(* PLC project Sem nome, Desconhecido Sem nome 1 *)
(* stored: creationDateTime 2025-09-02T10:17:35, modificationDateTime 2025-09-05T09:58:23 *)

PROGRAM program0
  VAR
    HighSensor AT %IX100.0 : BOOL;
    LowSensor AT %IX100.1 : BOOL;
    PalletSensor AT %IX100.2 : BOOL;
    Loaded AT %IX100.3 : BOOL;
    AtLeftEntry AT %IX100.4 : BOOL;
    AtLeftExit AT %IX100.5 : BOOL;
    AtRightEntry AT %IX100.6 : BOOL;
    AtRightExit AT %IX100.7 : BOOL;
    Start AT %IX100.8 : BOOL;
    Reset AT %IX100.9 : BOOL;
    Stop AT %IX100.10 : BOOL;
    EmergencyStop AT %IX100.11 : BOOL;
    Auto AT %IX100.12 : BOOL;
    ConveyorEntry AT %QX100.0 : BOOL;
    Load AT %QX100.1 : BOOL;
    Unload AT %QX100.2 : BOOL;
    TransferLeft AT %QX100.3 : BOOL;
    TransferRight AT %QX100.4 : BOOL;
    ConveyorLeft AT %QX100.5 : BOOL;
    ConveyorRight AT %QX100.6 : BOOL;
    StartLight AT %QX100.7 : BOOL;
    ResetLight AT %QX100.8 : BOOL;
    StopLight AT %QX100.9 : BOOL;
  END_VAR
  VAR
    MemoryRight : BOOL;
    MemoryLeft : BOOL;
  END_VAR
  VAR
    Counter AT %QW100 : INT;
  END_VAR
  VAR
    CTU0 : CTU;
  END_VAR
  VAR  (* added by the conversion: wires and edge detectors of the diagram *)
    R_TRIG1 : R_TRIG;
  END_VAR

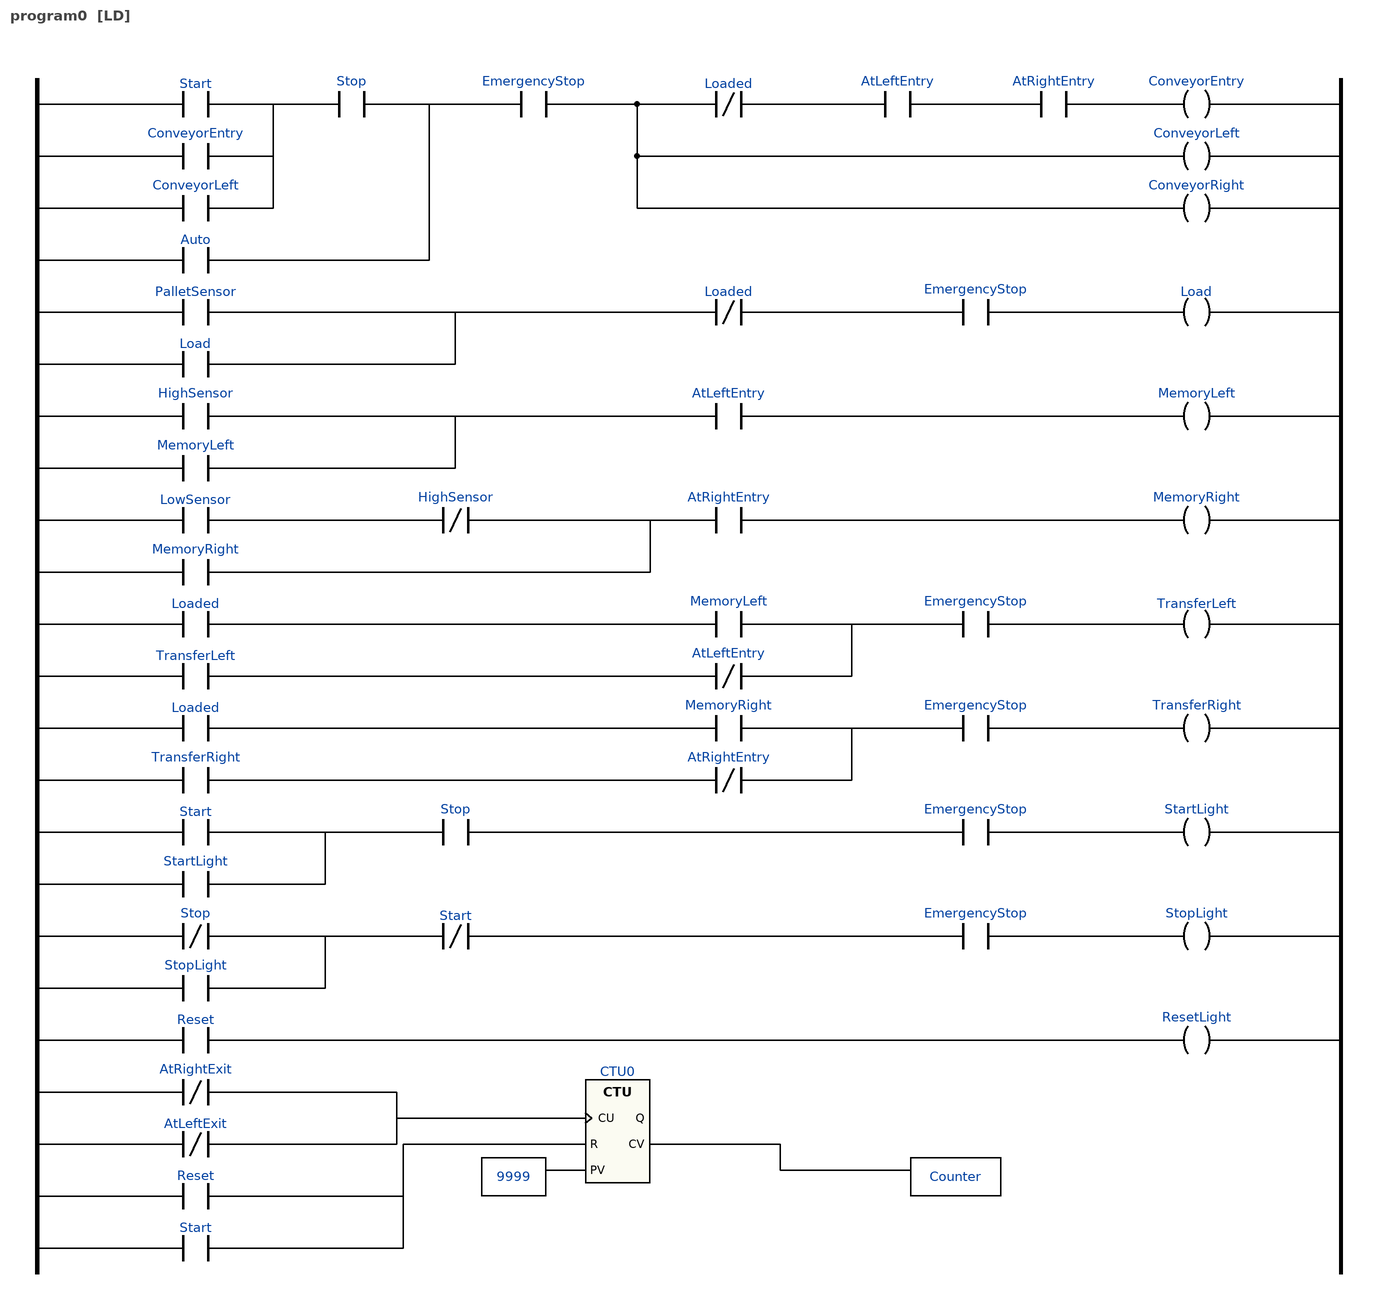
(* LD diagram, written out as Structured Text *)
ConveyorEntry := ((Start OR ConveyorEntry OR ConveyorLeft) AND Stop OR Auto) AND EmergencyStop AND NOT Loaded AND AtLeftEntry AND AtRightEntry;
ConveyorLeft := ((Start OR ConveyorEntry OR ConveyorLeft) AND Stop OR Auto) AND EmergencyStop;
ConveyorRight := ((Start OR ConveyorEntry OR ConveyorLeft) AND Stop OR Auto) AND EmergencyStop;
Load := (PalletSensor OR Load) AND NOT Loaded AND EmergencyStop;
MemoryLeft := (HighSensor OR MemoryLeft) AND AtLeftEntry;
MemoryRight := (MemoryRight OR LowSensor AND NOT HighSensor) AND AtRightEntry;
TransferLeft := (Loaded AND MemoryLeft OR TransferLeft AND NOT AtLeftEntry) AND EmergencyStop;
TransferRight := (Loaded AND MemoryRight OR TransferRight AND NOT AtRightEntry) AND EmergencyStop;
StartLight := (Start OR StartLight) AND Stop AND EmergencyStop;
StopLight := (NOT Stop OR StopLight) AND NOT Start AND EmergencyStop;
ResetLight := Reset;
R_TRIG1(CLK := NOT AtRightExit OR NOT AtLeftExit);
CTU0(CU := R_TRIG1.Q, R := Reset OR Start, PV := 9999);
Counter := CTU0.CV;
END_PROGRAM

CONFIGURATION Config0
  RESOURCE Res0 ON PLC
    TASK task0(INTERVAL := T#20ms, PRIORITY := 0);
    PROGRAM instance0 WITH task0 : program0;
  END_RESOURCE
END_CONFIGURATION
